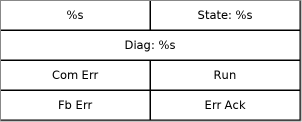
VISUALIZATION TplTsGroupExt  // 302x122
VAR_IN_OUT
	stGroupDiag					:FB_TwinSafeGroupExt;
END_VAR
(* End *)
    Rectangle (0,60 150x30), "Com Err", colour toggle: stGroupDiag.bComErr
    Rectangle (0,90 150x30), "Fb Err", colour toggle: stGroupDiag.bFbErr
    Rectangle (150,0 150x30), "State: %s", text variable: stGroupDiag.sState, colour toggle: stGroupDiag.sState = 'ERROR'
    Rectangle (150,60 150x30), "Run", colour toggle: stGroupDiag.bRun
    Rectangle (150,90 150x30), "Err Ack", colour toggle: stGroupDiag.bErrAck
    Rectangle (0,0 150x30), "%s", text variable: stGroupDiag.sName, colour toggle: stGroupDiag.sState = 'RUN'
    Rectangle (0,30 300x30), "Diag: %s", text variable: stGroupDiag.sDiag
END_VISUALIZATION

(* stored: Version 1.1.0.1, ProductVersion 3.1.4024.11
   Visu TplTsGroupExt: Id {b150be7e-2453-405c-81d7-6c63f17c8033} *)
